TYPE Request :
STRUCT
	Command			:UINT;		// Value according to the command table
	Data			:ARRAY[0..18] OF UINT := [0];		
END_STRUCT
END_TYPE

(* stored: Version 1.1.0.1
   DUT Request: Id {57bcae6b-3fd8-48d8-877c-3358049e8c58} *)
